Fanuc KAREL source: CA0105.KL

-- PROVISIONAL review KL for V1013-1; original PC SHA256 78799eb1776a5377a898f2f8384d34e232f70feeac38edb16269152df9024c5d
-- Incomplete behavior may be omitted. Consult companion uncertainty JSON. Do not deploy.
PROGRAM CA0105
%NOLOCKGROUP
BEGIN
  -- UNRESOLVED_PC offsets 0-1; opcodes 7B
  -- UNRESOLVED_PC offsets 6-18; opcodes 2D,9D,52,7F
  -- UNRESOLVED_PC offsets 23-27; opcodes 7F
  -- UNRESOLVED_PC offsets 32-39; opcodes 9C,23
  -- UNRESOLVED_PC offsets 44-51; opcodes 9D,23
  -- UNRESOLVED_PC offsets 56-67; opcodes 2E,23
  -- UNRESOLVED_PC offsets 72-79; opcodes 9D,23
  -- UNRESOLVED_PC offsets 84-93; opcodes 3F,75
  -- UNRESOLVED_PC offsets 98-112; opcodes 2E,22,9D,33,35
  -- UNRESOLVED_PC offsets 117-131; opcodes 2E,22,9D,33,35
  -- UNRESOLVED_PC offsets 136-151; opcodes 2E,22,32,35
  -- UNRESOLVED_PC offsets 156-171; opcodes 2E,22,32,35
  -- UNRESOLVED_PC offsets 176-192; opcodes 27,22,AA,23
  -- UNRESOLVED_PC offsets 197-201; opcodes 7F
END CA0105
